# EPICS StreamDevice protocol: rsfsxApp/Db/rsfsx.proto
#---------------------------------------------------------------------
# Title      : Rohde & Schwarz FSL Spectrum Analyzer Epics Protocol File
# Project    :
#---------------------------------------------------------------------
# File       : rsfsl.proto
# Author     : Leticia Garcez Capovilla
# Company    : Brazilian Synchrotron Light Laboratory, LNLS/CNPEM
# Created    : 2018-03-19
# Last update: 2018-04-04
#---------------------------------------------------------------------
# Description:
#
# Defines protocol to use the device as a StreamDevice IOC in EPICS
#
#---------------------------------------------------------------------
# Copyright (c) 2018 Brazilian Synchrotron Light Laboratory, LNLS/CNPEM
#
# This program is free software: you can redistribute it and/or
# modify it under the terms of the GNU Lesser General Public License
# as published by the Free Software Foundation, either version 3 of
# the License, or (at your option) any later version.
#
# This program is distributed in the hope that it will be useful, but
# WITHOUT ANY WARRANTY; without even the implied warranty of
# MERCHANTABILITY or FITNESS FOR A PARTICULAR PURPOSE.  See the GNU
# Lesser General Public License for more details.
#
# You should have received a copy of the GNU Lesser General Public
# License along with this program. If not, see
# <http://www.gnu.org/licenses/>.
#---------------------------------------------------------------------
# Revisions  :
# Date        	Version  	Author          	Description
# 2018-mar-19	1.0      	leticiagcapovilla       Created
# 2018-apr-04	1.0		leticiagcapovilla	Updated
#---------------------------------------------------------------------

######################################################################
#
# Variable declaration
#
GLOBAL_TIMEOUT = 5000;

######################################################################
#
# Communication setup
#
OutTerminator = CR LF;
InTerminator = LF;
ExtraInput = Ignore;
MaxInput = 576018;
WriteTimeout = ${GLOBAL_TIMEOUT};
ReadTimeout = ${GLOBAL_TIMEOUT};
ReplyTimeout = ${GLOBAL_TIMEOUT};
Separator = ",";
#
#
######################################################################
# Reference Level

inRefLvl {
    out "DISP:WIND:TRAC:Y:SCAL:RLEV?";
    in "%f";
}

outRefLvl {
    out "DISP:WIND:TRAC:Y:SCAL:RLEV %f";
    @init { inRefLvl; };
}

######################################################################
# Reference Level Offset

inRefOff {
    out "DISP:WIND:TRAC:Y:SCAL:RLEV:OFFS?";
    in "%f";
}

outRefOff {
    out "DISP:WIND:TRAC:Y:SCAL:RLEV:OFFS %f";
    @init { inRefOff; };
}

######################################################################
# Enable Continuous Sweep Mode

inEnblContSwe {
    out "INIT:CONT?";
    in "%i";
}

outEnblContSwe {
    out "INIT:CONT %{OFF|ON}";
    @init { inEnblContSwe; };
}

######################################################################
# Sweep Points Number (MIN 101; MAX 32001)

inSwePts {
    out "SENS:SWE:POIN?";
    in "%i";
}

outSwePts {
    out "SENS:SWE:POIN %i";
    @init { inSwePts; };
}

######################################################################
# Sweep time

inSweTime {
    out "SENS:SWE:TIME?";
    in "%f";
}

outSweTime {
    out "SENS:SWE:TIME %f";
    @init { inSweTime; };
}

######################################################################
# Enable/Disable automatic coupling of the sweep time to the
# frequency span and bandwidth settings

inEnblSweTimeAuto {
    out "SENS:SWE:TIME:AUTO?";
    in "%i";
}

outEnblSweTimeAuto {
    out "SENS:SWE:TIME:AUTO %{OFF|ON}";
    @init { inEnblSweTimeAuto; };
}

######################################################################
# Type of display and evaluation of the trace

inTraceMode {
    out "DISP:WIND:TRAC1:MODE?";
    in "%{WRIT|VIEW|AVER|MAXH|MINH|BLANK}";
}

outTraceMode {
    out "DISP:WIND:TRAC1:MODE %{WRIT|VIEW|AVER|MAXH|MINH|BLANK}";
    @init { inTraceMode; };
}

######################################################################
# Center Frequency

inFrqCent {
    out "SENS:FREQ:CENT?";
    in "%f";
}

outFrqCent {
    out "SENS:FREQ:CENT %f";
    @init { inFrqCent; };
}

######################################################################
# Frequency Step

inFreqStep {
    out "SENS:FREQ:CENT:STEP?";
    in "%f";
}

outFreqStep {
    out "SENS:FREQ:CENT:STEP %f";
    @init { inFreqStep; };
}

######################################################################
# Frequency Step Link

inStepLink {
    out "SENS:FREQ:CENT:STEP:LINK?";
    in "%s";
}

outStepLink {
    out "SENS:FREQ:CENT:STEP:LINK %{SPAN|RBW|OFF}";
    @init { inStepLink; };
}

######################################################################
# Enable/Disable Auto Frequency Step (step coupled to span)

inAutoStep {
    out "SENS:FREQ:CENT:STEP:AUTO?";
    in "%i";
}

outAutoStep {
    out "SENS:FREQ:CENT:STEP:AUTO %{OFF|ON}";
    @init { inAutoStep; };
}

######################################################################
# Frequency Span

inFrqSpan {
    out "SENS:FREQ:SPAN?";
    in "%f";
}

outFrqSpan {
    out "SENS:FREQ:SPAN %f";
    @init { inFrqSpan; };
}

#####################################################################
# Start Frequency

inFrqStart {
    out "SENS:FREQ:STAR?";
    in "%f";
}

outFrqStart {
    out "SENS:FREQ:STAR %f";
    @init { inFrqStart; };
}

######################################################################
# Stop Frequency

inFrqStop {
    out "SENS:FREQ:STOP?";
    in "%f";
}

outFrqStop {
    out "SENS:FREQ:STOP %f";
    @init { inFrqStop; };
}

######################################################################
# Enable/Disable Markers (1-4)

inEnblMark1 {
    out "CALC:MARK1:STAT?";
    in "%i";
}

outEnblMark1 {
    out "CALC:MARK1:STAT %i";
    @init { inEnblMark1; };
}

inEnblMark2 {
    out "CALC:MARK2:STAT?";
    in "%i";
}

outEnblMark2 {
    out "CALC:MARK2:STAT %i";
    @init { inEnblMark2; };
}

outOnOffM2 {
    out "CALC:MARK2:STAT %i";
}

inEnblMark3 {
    out "CALC:MARK3:STAT?";
    in "%i";
}

outEnblMark3 {
    out "CALC:MARK3:STAT %i";
    @init { inEnblMark3; };
}

outOnOffM3 {
    out "CALC:MARK3:STAT %i";
}

inEnblMark4 {
    out "CALC:MARK4:STAT?";
    in "%i";
}

outEnblMark4 {
    out "CALC:MARK4:STAT %i";
    @init { inEnblMark4; };
}

outOnOffM4 {
    out "CALC:MARK4:STAT %i";
}

######################################################################
# Markers X Values

inMarkX1 {
    out "CALC:MARK1:X?";
    in "%f";
}

outMarkX1 {
    out "CALC:MARK1:X %f";
}

inMarkX2 {
    out "CALC:MARK2:X?";
    in "%f";
}

outMarkX2 {
    out "CALC:MARK2:X %f";
}

inMarkX3 {
    out "CALC:MARK3:X?";
    in "%f";
}

outMarkX3 {
    out "CALC:MARK3:X %f";
}

inMarkX4 {
    out "CALC:MARK4:X?";
    in "%f";
}

outMarkX4 {
    out "CALC:MARK4:X %f";
}

######################################################################
# Enable Marker Frequency Counter (only available for Marker1)

inEnblMarkCount {
    out "CALC:MARK:COUN?";
    in "%i";
}

outEnblMarkCount {
    out "CALC:MARK:COUN %i";
}

#######################################################################
## Enable local oscillator supression for peak search
#
#inEnblLocalOscSupr {
#    out "CALC:MARK:LOEX?";
#    in "%i";
#}
#
#outEnblLocalOscSupr {
#    out "CALC:MARK:LOEX %i";
#}
#
#######################################################################
# Enable automatic peak search (only available for Marker1)

inEnblMaxAuto {
    out "CALC:MARK:MAX:AUTO?";
    in "%i";
}

outEnblMaxAuto {
    out "CALC:MARK:MAX:AUTO %{OFF|ON}";
}

######################################################################
# Enable automatic peak search (only available for Marker1)

inEnblMinAuto {
    out "CALC:MARK:MIN:AUTO?";
    in "%i";
}

outEnblMinAuto {
    out "CALC:MARK:MIN:AUTO %{OFF|ON}";
}

######################################################################
# Define the peak excursion

inMarkPExcursion {
    out "CALC:MARK:PEXC?";
    in "%f";
}

outMarkPExcursion {
    out "CALC:MARK:PEXC %f";
}

######################################################################
# Enable/Disable limited search range

inEnblMarkLimit {
    out "CALC:MARK:X:SLIM:STAT?";
    in "%i";
}

outEnblMarkLimit {
    out "CALC:MARK:X:SLIM:STAT %{OFF|ON}";
}

######################################################################
# Left limit for the search range

inMarkLimitLeft {
    out "CALC:MARK:X:SLIM:LEFT?";
    in "%f";
}

outMarkLimitLeft {
    out "CALC:MARK:X:SLIM:LEFT %f";
}

######################################################################
# Right limit for the search range

inMarkLimitRight {
    out "CALC:MARK:X:SLIM:RIGHT?";
    in "%f";
}

outMarkLimitRight {
    out "CALC:MARK:X:SLIM:RIGHT %f";
}

######################################################################
# Enable/Disable Delta Markers (1-4)

inEnblDMark1 {
    out "CALC:DELT1:STAT?";
    in "%i";
}

outEnblDMark1 {
    out "CALC:DELT1:STAT %i";
    @init { inEnblDMark1; };
}

outOnOffDM1 {
    out "CALC:DELT1:STAT %i";
}

inEnblDMark2 {
    out "CALC:DELT2:STAT?";
    in "%i";
}

outEnblDMark2 {
    out "CALC:DELT2:STAT %i";
    @init { inEnblDMark2; };
}

outOnOffDM2 {
    out "CALC:DELT2:STAT %i";
}

inEnblDMark3 {
    out "CALC:DELT3:STAT?";
    in "%i";
}

outEnblDMark3 {
    out "CALC:DELT3:STAT %i";
    @init { inEnblDMark3; };
}

outOnOffDM3 {
    out "CALC:DELT3:STAT %i";
}

inEnblDMark4 {
    out "CALC:DELT4:STAT?";
    in "%i";
}

outEnblDMark4 {
    out "CALC:DELT4:STAT %i";
    @init { inEnblDMark4; };
}

outOnOffDM4 {
    out "CALC:DELT4:STAT %i";
}

######################################################################
# Delta Markers X Values

inDMarkX1 {
    out "CALC:DELT1:X?";
    in "%f";
}

outDMarkX1 {
    out "CALC:DELT1:X %f";
}

inDMarkX2 {
    out "CALC:DELT2:X?";
    in "%f";
}

outDMarkX2 {
    out "CALC:DELT2:X %f";
}

inDMarkX3 {
    out "CALC:DELT3:X?";
    in "%f";
}

outDMarkX3 {
    out "CALC:DELT3:X %f";
}

inDMarkX4 {
    out "CALC:DELT4:X?";
    in "%f";
}

outDMarkX4 {
    out "CALC:DELT4:X %f";
}

#####################################################################
# State of tracking generator output

inEnblOut {
    out "OUTP:STAT?";
    in "%i";
}

outEnblOut {
    out "OUTP:STAT %{OFF|ON}";
    @init { inEnblOut; };
}

#######################################################################
## Enable/Disable Tracking Generator Normalization of the measurement
## results
#
#inEnblOutCorrect {
#    out "SENS:CORR:STAT?";
#    in "%i";
#}
#
#outEnblOutCorrect {
#    out "SENS:CORR:STAT %{OFF|ON}";
#}
#
######################################################################
# Input Attenuator Value

inAttIn {
    out "INP:ATT?";
    in "%i";
}

outAttIn {
    out "INP:ATT %i";
}

######################################################################
# Enable/Disable automatic coupling of the input attenuation to the
# reference level

inEnblAttAuto {
    out "INP:ATT:AUTO?";
    in 	"%i";
}

outEnblAttAuto {
    out "INP:ATT:AUTO %{OFF|ON}";
}

######################################################################
## Enable/Disable Input Preamplifier - Only available on R&S FSL-B22
#
#inEnblPreamp {
#    out "INP:GAIN:STAT?";
#    in "%i";
#}
#
#outEnblPreamp {
#    out "INP:GAIN:STAT %i";
#}
#
######################################################################
# Instruments Nominal input impedance

inImpdIn {
    out "INP:IMP?";
    in "%{50|75}";
}

outImpdIn {
    out "INP:IMP %{50|75}";
}

######################################################################
# Oscillator Reference

inRoscSrc {
    out "SOUR:EXT:ROSC:SOUR?";
    in "%{INT|EXT}";
}

outRoscSrc {
    out "SOUR:EXT:ROSC:SOUR %{INT|EXT}";
}

######################################################################
# Tracking Generator Level

inLvlOut {
    out "SOUR:POW:LEV:IMM:AMPL?";
    in "%f";
}

outLvlOut {
    out "SOUR:POW:LEV:IMM:AMPL %f";
}

######################################################################
# Tracking Generator Offset Level

inLvlOutOffset {
    out "SOUR:POW:LEV:IMM:OFFS?";
    in "%f";
}

outLvlOutOffset {
    out "SOUR:POW:LEV:IMM:OFFS %f";
}

######################################################################
# Resolution Bandwidth

inRbw {
    out "SENS:BWID:RES?";
    in "%i";
}

outRbw {
    out "SENS:BWID:RES %i";
}

######################################################################
# Video Bandwidth

inVbw {
    out "SENS:BWID:VID?";
    in "%i";
}

outVbw {
    out "SENS:BWID:VID %i";
}

######################################################################
# Enable/Disable automatic coupling of the video bandwidth to the
# resolution bandwidth

inEnblVbwAuto {
    out "SENS:BWID:VID:AUTO?";
    in "%i";
}

outEnblVbwAuto {
    out "SENS:BWID:VID:AUTO %{OFF|ON}";
}

######################################################################
# Select Filter Type

inFiltType {
    out "SENS:BWID:RES:TYPE?";
    in "%s";
}

outFiltType {
    out "SENS:BWID:RES:TYPE %{NORM|FFT|CFIL|RRC|PULS}";
}

######################################################################
# Select Detector Type Manually

inDetecType {
    out "SENS:DET:FUNC?";
    in "%s";
}

outDetecType {
    out "SENS:DET:FUNC %{APE|NEG|POS|SAMP|RMS|AVER|QPE}";
}

######################################################################
# Enable/Disable spectrogram measurement (SPECM, option K14)

inEnblSpec {
    out "CALC:SPEC:STAT?";
    in "%i";
}

outEnblSpec {
    out "CALC:SPEC:STAT %{OFF|ON}";
}

######################################################################
# Enable/Disable continuous sweep measurement (SPECM, option K14)

inEnblSweCont {
    out "INIT:CONT?";
    in "%i";
}

outEnblSweCont {
    out "INIT:CONT %{ON|OFF}";
}

######################################################################
# Enable/Disable delete of previous measurement

inEnblDelMeas {
    out "CALC:SPEC:CONT?";
    in "%i";
}

outEnblDelMeas {
    out "CALC:SPEC:CONT %{OFF|ON}";
}

######################################################################
# Number of frames recorded (SPECM, Opt. K14)

inSpecFrameCount {
    out "CALC:SPEC:FRAM:COUN?";
    in "%f";
}

outSpecFrameCount {
    out "CALC:SPEC:FRAM:COUN %f";
}

######################################################################
# Frame selection (SPECM, Opt. K14)

inSpecFrame {
    out "CALC:SPEC:FRAM:SEL?";
    in "%f";
}

outSpecFrame {
    out "CALC:SPEC:FRAM:SEL %f";
}

######################################################################
# History Depth

inSpecBuffSize {
    out "CALC:SPEC:HDEP?";
    in "%f";
}

outSpecBuffSize {
    out "CALC:SPEC:HDEP %f";
}

######################################################################
########################### MONITOR ##################################
######################################################################
# Get identification

inIdn {
    out "*IDN?";
    in "%s";
}

######################################################################
# Markers Y Values

monMarkY1 {
    out "CALC:MARK1:Y?";
    in "%f";
}

monMarkY2 {
    out "CALC:MARK2:Y?";
    in "%f";
}

monMarkY3 {
    out "CALC:MARK3:Y?";
    in "%f";
}

monMarkY4 {
    out "CALC:MARK4:Y?";
    in "%f";
}

######################################################################
# Delta Markers Y Values

monDMarkY1 {
    out "CALC:DELT1:Y?";
    in "%f";
}

monDMarkY2 {
    out "CALC:DELT2:Y?";
    in "%f";
}

monDMarkY3 {
    out "CALC:DELT3:Y?";
    in "%f";
}

monDMarkY4 {
    out "CALC:DELT4:Y?";
    in "%f";
}

######################################################################
# Queries the result of the markers frequency count (only available for Marker1)

monMarkCount {
    out "CALC:MARK:COUN:FREQ?";
    in "%f";
}

######################################################################
# Trace Data (one waveform per sweep, retrieves level information)

monTrace {
    out "TRAC? TRACE1";
    in "%f";
}

######################################################################
# Level Data for Spectrogram Acquisition

monSpec {
    out "TRAC? TRACE1";
    in "%f";
}

######################################################################
# Data Format (always use ASCII format)

outDataFormat {
    out "FORM:DATA ASC";
    @init { outDataFormat; };
}

######################################################################
########################### COMMAND ##################################
######################################################################
# Reset to default state
cmdRst {
    out "%{|*RST; *WAI}";
}

######################################################################
# Set Markers to Max Peak on Trace (1-4)

cmdMarkMax1 {
    out "%{|CALC:MARK1:MAX:PEAK}";
}

cmdMarkMax2 {
    out "%{|CALC:MARK2:MAX:PEAK}";
}

cmdMarkMax3 {
    out "%{|CALC:MARK3:MAX:PEAK}";
}

cmdMarkMax4 {
    out "%{|CALC:MARK4:MAX:PEAK}";
}

######################################################################
# Set Delta Markers to Max Peak on Trace (1-4)

cmdDMarkMax1 {
    out "%{|CALC:DELT1:MAX:PEAK}";
}

cmdDMarkMax2 {
    out "%{|CALC:DELT2:MAX:PEAK}";
}

cmdDMarkMax3 {
    out "%{|CALC:DELT3:MAX:PEAK}";
}

cmdDMarkMax4 {
    out "%{|CALC:DELT4:MAX:PEAK}";
}

######################################################################
# Turn all markers off

cmdMarkAOff {
    out "%{|CALC:MARK:AOFF}";
}

######################################################################
# Position the marker to the next smaller maximium value to the left
# of the current value (1-4)

cmdMarkMaxLeft1 {
    out "%{|CALC:MARK1:MAX:LEFT}";
}

cmdMarkMaxLeft2 {
    out "%{|CALC:MARK2:MAX:LEFT}";
}

cmdMarkMaxLeft3 {
    out "%{|CALC:MARK3:MAX:LEFT}";
}

cmdMarkMaxLeft4 {
    out "%{|CALC:MARK4:MAX:LEFT}";
}

######################################################################
# Position the delta marker to the next smaller maximium value to the left
# of the current value (1-4)

cmdDMarkMaxLeft1 {
    out "%{|CALC:DELT1:MAX:LEFT}";
}

cmdDMarkMaxLeft2 {
    out "%{|CALC:DELT2:MAX:LEFT}";
}

cmdDMarkMaxLeft3 {
    out "%{|CALC:DELT3:MAX:LEFT}";
}

cmdDMarkMaxLeft4 {
    out "%{|CALC:DELT4:MAX:LEFT}";
}

######################################################################
# Position the marker to the next smaller minimium value to the left
# of the current value (1-4)

cmdMarkMinLeft1 {
    out "%{|CALC:MARK1:MIN:LEFT}";
}

cmdMarkMinLeft2 {
    out "%{|CALC:MARK2:MIN:LEFT}";
}

cmdMarkMinLeft3 {
    out "%{|CALC:MARK3:MIN:LEFT}";
}

cmdMarkMinLeft4 {
    out "%{|CALC:MARK4:MIN:LEFT}";
}

######################################################################
# Position the delta marker to the next smaller minimium value to the left
# of the current value (1-4)

cmdDMarkMinLeft1 {
    out "%{|CALC:DELT1:MIN:LEFT}";
}

cmdDMarkMinLeft2 {
    out "%{|CALC:DELT2:MIN:LEFT}";
}

cmdDMarkMinLeft3 {
    out "%{|CALC:DELT3:MIN:LEFT}";
}

cmdDMarkMinLeft4 {
    out "%{|CALC:DELT4:MIN:LEFT}";
}

######################################################################
# Position the marker to the next smaller maximium value of the
# corresponding trace (1-4)

cmdMarkMaxNext1 {
    out "%{|CALC:MARK1:MAX:NEXT}";
}

cmdMarkMaxNext2 {
    out "%{|CALC:MARK2:MAX:NEXT}";
}

cmdMarkMaxNext3 {
    out "%{|CALC:MARK3:MAX:NEXT}";
}

cmdMarkMaxNext4 {
    out "%{|CALC:MARK4:MAX:NEXT}";
}

######################################################################
# Position the delta marker to the next smaller maximium value of the
# corresponding trace (1-4)

cmdDMarkMaxNext1 {
    out "%{|CALC:DELT1:MAX:NEXT}";
}

cmdDMarkMaxNext2 {
    out "%{|CALC:DELT2:MAX:NEXT}";
}

cmdDMarkMaxNext3 {
    out "%{|CALC:DELT3:MAX:NEXT}";
}

cmdDMarkMaxNext4 {
    out "%{|CALC:DELT4:MAX:NEXT}";
}

######################################################################
# Position the marker to the next smaller minimium value of the
# corresponding trace (1-4)

cmdMarkMinNext1 {
    out "%{|CALC:MARK1:MIN:NEXT}";
}

cmdMarkMinNext2 {
    out "%{|CALC:MARK2:MIN:NEXT}";
}

cmdMarkMinNext3 {
    out "%{|CALC:MARK3:MIN:NEXT}";
}

cmdMarkMinNext4 {
    out "%{|CALC:MARK4:MIN:NEXT}";
}

######################################################################
# Position the delta marker to the next smaller minimium value of the
# corresponding trace (1-4)

cmdDMarkMinNext1 {
    out "%{|CALC:DELT1:MIN:NEXT}";
}

cmdDMarkMinNext2 {
    out "%{|CALC:DELT2:MIN:NEXT}";
}

cmdDMarkMinNext3 {
    out "%{|CALC:DELT3:MIN:NEXT}";
}

cmdDMarkMinNext4 {
    out "%{|CALC:DELT4:MIN:NEXT}";
}

#####################################################################
# Position the marker to the next smaller maximium value to the right
# of the current value (1-4)

cmdMarkMaxRight1 {
    out "%{|CALC:MARK1:MAX:RIGHT}";
}

cmdMarkMaxRight2 {
    out "%{|CALC:MARK2:MAX:RIGHT}";
}

cmdMarkMaxRight3 {
    out "%{|CALC:MARK3:MAX:RIGHT}";
}

cmdMarkMaxRight4 {
    out "%{|CALC:MARK4:MAX:RIGHT}";
}

#####################################################################
# Position the delta marker to the next smaller maximium value to the right
# of the current value (1-4)

cmdDMarkMaxRight1 {
    out "%{|CALC:DELT1:MAX:RIGHT}";
}

cmdDMarkMaxRight2 {
    out "%{|CALC:DELT2:MAX:RIGHT}";
}

cmdDMarkMaxRight3 {
    out "%{|CALC:DELT3:MAX:RIGHT}";
}

cmdDMarkMaxRight4 {
    out "%{|CALC:DELT4:MAX:RIGHT}";
}

#####################################################################
# Position the marker to the next smaller minimium value to the right
# of the current value (1-4)

cmdMarkMinRight1 {
    out "%{|CALC:MARK1:MIN:RIGHT}";
}

cmdMarkMinRight2 {
    out "%{|CALC:MARK2:MIN:RIGHT}";
}

cmdMarkMinRight3 {
    out "%{|CALC:MARK3:MIN:RIGHT}";
}

cmdMarkMinRight4 {
    out "%{|CALC:MARK4:MIN:RIGHT}";
}

#####################################################################
# Position the delta marker to the next smaller minimium value to the right
# of the current value (1-4)

cmdDMarkMinRight1 {
    out "%{|CALC:DELT1:MIN:RIGHT}";
}

cmdDMarkMinRight2 {
    out "%{|CALC:DELT2:MIN:RIGHT}";
}

cmdDMarkMinRight3 {
    out "%{|CALC:DELT3:MIN:RIGHT}";
}

cmdDMarkMinRight4 {
    out "%{|CALC:DELT4:MIN:RIGHT}";
}

#####################################################################
# Set Markers to Min Peak on Trace (1-4)

cmdMarkMin1 {
    out "%{|CALC:MARK1:MIN:PEAK}";
}

cmdMarkMin2 {
    out "%{|CALC:MARK2:MIN:PEAK}";
}

cmdMarkMin3 {
    out "%{|CALC:MARK3:MIN:PEAK}";
}

cmdMarkMin4 {
    out "%{|CALC:MARK4:MIN:PEAK}";
}

#####################################################################
# Set Delta Markers to Min Peak on Trace (1-4)

cmdDMarkMin1 {
    out "%{|CALC:DELT1:MIN:PEAK}";
}

cmdDMarkMin2 {
    out "%{|CALC:DELT2:MIN:PEAK}";
}

cmdDMarkMin3 {
    out "%{|CALC:DELT3:MIN:PEAK}";
}

cmdDMarkMin4 {
    out "%{|CALC:DELT4:MIN:PEAK}";
}

######################################################################
# Switch off all Delta Markers

cmdDMarkAOff {
    out "%{|CALC:DELT:AOFF}";
}

#######################################################################
## Initiate a new measurement sequence
#
#cmdInitMeas {
#    out "%{|INIT:IMM}";
#}
#
#######################################################################
## Continue a stopped measurement in single sweep mode
#
#cmdConMeas {
#    out "%{|INIT:CONM}";
#}
#
#######################################################################
## Start a Spectrum Emission Mask Measurement
#
#cmdSpecEmisMeas {
#    out "%{|INIT:ESP}";
#}
#
#######################################################################
## Start a Spurious Emissions Measurement
#
#cmdSpurEmisMeas {
#    out "%{|INIT:SPUR}";
#}
#

######################################################################
# Clean spectrogram and history buffer

cmdCleanSpec {
    out "CALC:SPEC:CLE:IMM";
}

######################################################################
############################## SAVE ##################################
######################################################################
# IQ Data

inIQ {
    Separator=",";
    out "INIT:CONT OFF";
    out "TRAC:IQ:STAT ON";
    out "TRAC:IQ:SET NORM,10 MHz,32 MHz,IMM,POS,0,10";
    out "TRAC:IQ:DATA?";
    in "%E";
}
